// TIA Portal project "BitToWord" (V16)

(* hardware
DEVICE "S71500/ET200MP station_1"  S7-1500 station
   slot 0: "Rail_0"  Rack  6ES7 590-1***0-0AA0
   slot 1: "PLC_1"  CPU 1511T-1 PN  6ES7 511-1TK01-0AB0  V2.8
      slot 3: "CPU display_1"  6ES7591-1AA00-0AA0
      slot 32768: "PROFINET interface_1"  X1
         slot 32769: "Port_1"  X1 P1
         slot 32770: "Port_2"  X1 P2
      slot 34817: "Virtual CP interface port_1"  Virtual CP interface port  Virtual CP interface port
*)

// ===== PLC "PLC_1"  CPU 1511T-1 PN =====

VAR_GLOBAL   // PLC tag table "Default tag table"
   "word_out" AT %MW0 : Word;
END_VAR

DATA_BLOCK "BitToWord_DB"   // DB1
{ S7_Optimized_Access := 'TRUE' }
VERSION : 0.1
// stored: InstanceOfName BitToWord
"BitToWord"
BEGIN
END_DATA_BLOCK

DATA_BLOCK "Bool_DB"   // DB2
{ S7_Optimized_Access := 'TRUE' }
VERSION : 0.1
   VAR
      Header : ArrayDBHeader;
      THIS : Array[0..15] of Bool;
   END_VAR
BEGIN
   Header.LowerBound := 0;
   Header.UpperBound := 15;
   Header.Elements := 16;
   Header.PaddedSize := 1;
   Header.ElementSize := 1;
   THIS[0] := 1;
   THIS[1] := 1;
   THIS[2] := 1;
   THIS[15] := 1;
   THIS[3] := 1;
   THIS[4] := 1;
   THIS[5] := 1;
   THIS[6] := 1;
   THIS[7] := 1;
   THIS[8] := 1;
   THIS[9] := 1;
   THIS[10] := 1;
   THIS[11] := 1;
   THIS[12] := 1;
   THIS[13] := 1;
   THIS[14] := 1;
END_DATA_BLOCK

FUNCTION_BLOCK "BitToWord"   // FB1, LAD
{ S7_Optimized_Access := 'TRUE' }
VERSION : 0.1
   VAR_INPUT
      in1 : Bool;
      in2 : Bool;
      in3 : Bool;
      in4 : Bool;
      in5 : Bool;
      in6 : Bool;
      in7 : Bool;
      in8 : Bool;
      in9 : Bool;
      in10 : Bool;
      in11 : Bool;
      in12 : Bool;
      in13 : Bool;
      in14 : Bool;
      in15 : Bool;
      in16 : Bool;
   END_VAR
   VAR_OUTPUT
      outWord : Word;
   END_VAR
   VAR
      bInput_word : Word;
      bool_array AT bInput_word : Array[0..15] of Bool;
   END_VAR
BEGIN

REGION Network 1
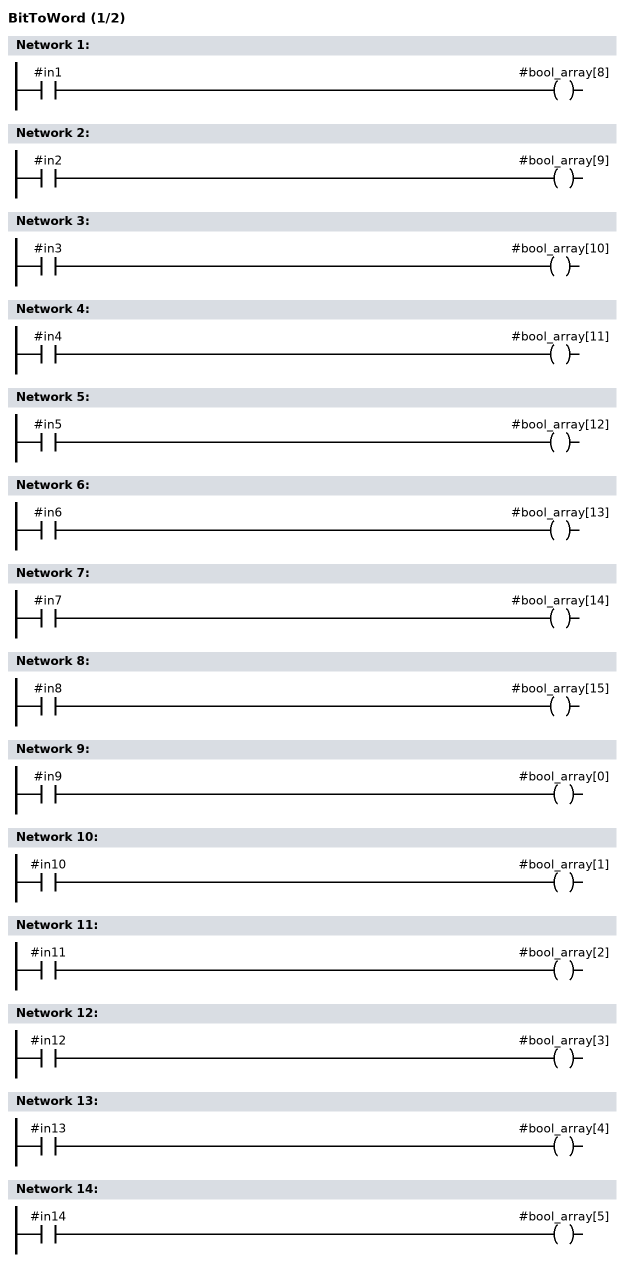
   RUNG wire#powerrail
      Contact( #in1 )
      Coil( #bool_array[8] )
   END_RUNG
   // the same network as SCL:
   #bool_array[8] := #in1;
END_REGION

REGION Network 2
   RUNG wire#powerrail
      Contact( #in2 )
      Coil( #bool_array[9] )
   END_RUNG
   // the same network as SCL:
   #bool_array[9] := #in2;
END_REGION

REGION Network 3
   RUNG wire#powerrail
      Contact( #in3 )
      Coil( #bool_array[10] )
   END_RUNG
   // the same network as SCL:
   #bool_array[10] := #in3;
END_REGION

REGION Network 4
   RUNG wire#powerrail
      Contact( #in4 )
      Coil( #bool_array[11] )
   END_RUNG
   // the same network as SCL:
   #bool_array[11] := #in4;
END_REGION

REGION Network 5
   RUNG wire#powerrail
      Contact( #in5 )
      Coil( #bool_array[12] )
   END_RUNG
   // the same network as SCL:
   #bool_array[12] := #in5;
END_REGION

REGION Network 6
   RUNG wire#powerrail
      Contact( #in6 )
      Coil( #bool_array[13] )
   END_RUNG
   // the same network as SCL:
   #bool_array[13] := #in6;
END_REGION

REGION Network 7
   RUNG wire#powerrail
      Contact( #in7 )
      Coil( #bool_array[14] )
   END_RUNG
   // the same network as SCL:
   #bool_array[14] := #in7;
END_REGION

REGION Network 8
   RUNG wire#powerrail
      Contact( #in8 )
      Coil( #bool_array[15] )
   END_RUNG
   // the same network as SCL:
   #bool_array[15] := #in8;
END_REGION

REGION Network 9
   RUNG wire#powerrail
      Contact( #in9 )
      Coil( #bool_array[0] )
   END_RUNG
   // the same network as SCL:
   #bool_array[0] := #in9;
END_REGION

REGION Network 10
   RUNG wire#powerrail
      Contact( #in10 )
      Coil( #bool_array[1] )
   END_RUNG
   // the same network as SCL:
   #bool_array[1] := #in10;
END_REGION

REGION Network 11
   RUNG wire#powerrail
      Contact( #in11 )
      Coil( #bool_array[2] )
   END_RUNG
   // the same network as SCL:
   #bool_array[2] := #in11;
END_REGION

REGION Network 12
   RUNG wire#powerrail
      Contact( #in12 )
      Coil( #bool_array[3] )
   END_RUNG
   // the same network as SCL:
   #bool_array[3] := #in12;
END_REGION

REGION Network 13
   RUNG wire#powerrail
      Contact( #in13 )
      Coil( #bool_array[4] )
   END_RUNG
   // the same network as SCL:
   #bool_array[4] := #in13;
END_REGION

REGION Network 14
   RUNG wire#powerrail
      Contact( #in14 )
      Coil( #bool_array[5] )
   END_RUNG
   // the same network as SCL:
   #bool_array[5] := #in14;
END_REGION

REGION Network 15
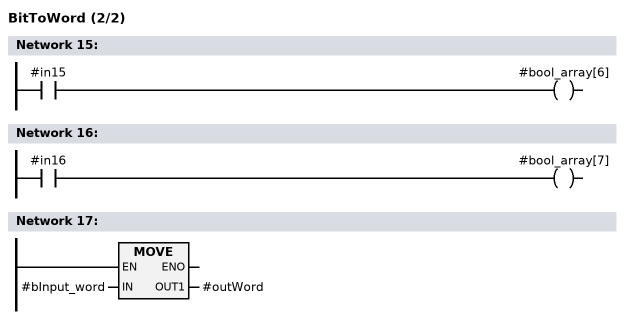
   RUNG wire#powerrail
      Contact( #in15 )
      Coil( #bool_array[6] )
   END_RUNG
   // the same network as SCL:
   #bool_array[6] := #in15;
END_REGION

REGION Network 16
   RUNG wire#powerrail
      Contact( #in16 )
      Coil( #bool_array[7] )
   END_RUNG
   // the same network as SCL:
   #bool_array[7] := #in16;
END_REGION

REGION Network 17
   RUNG wire#powerrail
      Move(in := #bInput_word, out1 => #outWord)
   END_RUNG
   // the same network as SCL:
   #outWord := #bInput_word;
END_REGION
END_FUNCTION_BLOCK

ORGANIZATION_BLOCK "Main"   // OB1, LAD, ProgramCycle
TITLE = "Main Program Sweep (Cycle)"
{ S7_Optimized_Access := 'TRUE' }
VERSION : 0.1
   VAR_INPUT
      Initial_Call : Bool;   // Initial call of this OB
      Remanence : Bool;   // =True, if remanent data are available
   END_VAR
BEGIN

REGION Network 1
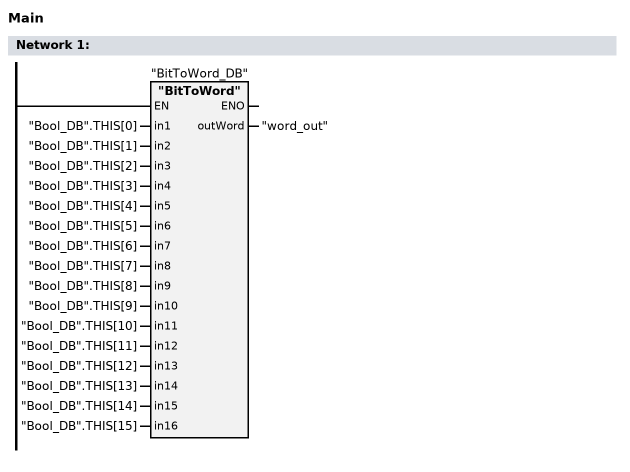
   RUNG wire#powerrail
      "BitToWord_DB"(in1 := "Bool_DB".THIS[0], in2 := "Bool_DB".THIS[1], in3 := "Bool_DB".THIS[2], in4 := "Bool_DB".THIS[3], in5 := "Bool_DB".THIS[4], in6 := "Bool_DB".THIS[5], in7 := "Bool_DB".THIS[6], in8 := "Bool_DB".THIS[7], in9 := "Bool_DB".THIS[8], in10 := "Bool_DB".THIS[9], in11 := "Bool_DB".THIS[10], in12 := "Bool_DB".THIS[11], in13 := "Bool_DB".THIS[12], in14 := "Bool_DB".THIS[13], in15 := "Bool_DB".THIS[14], in16 := "Bool_DB".THIS[15], outWord => "word_out")
   END_RUNG
   // the same network as SCL:
   "BitToWord_DB"(in1 := "Bool_DB".THIS[0],   // "BitToWord"
                  in2 := "Bool_DB".THIS[1],
                  in3 := "Bool_DB".THIS[2],
                  in4 := "Bool_DB".THIS[3],
                  in5 := "Bool_DB".THIS[4],
                  in6 := "Bool_DB".THIS[5],
                  in7 := "Bool_DB".THIS[6],
                  in8 := "Bool_DB".THIS[7],
                  in9 := "Bool_DB".THIS[8],
                  in10 := "Bool_DB".THIS[9],
                  in11 := "Bool_DB".THIS[10],
                  in12 := "Bool_DB".THIS[11],
                  in13 := "Bool_DB".THIS[12],
                  in14 := "Bool_DB".THIS[13],
                  in15 := "Bool_DB".THIS[14],
                  in16 := "Bool_DB".THIS[15],
                  outWord => "word_out");
END_REGION
END_ORGANIZATION_BLOCK